PROGRAM PRG_SmartHome
VAR
	HallRoom: FB_HallRoom;
END_VAR


	HallRoom(Lamp=> , Dimmer=> );

END_PROGRAM

(* stored: Version 1.1.0.1, ProductVersion 3.1.4024.12
   POU PRG_SmartHome: Id {3a9a704e-ac95-4023-9fa2-f778a7ebe871}, SpecialFunc None *)
